ABB RAPID module: EGM_test_UDP.mod

MODULE EGM_test_UDP

    VAR egmident egmID1;
    VAR egmstate egmSt1;

    CONST egm_minmax egm_minmax_lin1:=[-1,1]; !in mm
    CONST egm_minmax egm_minmax_rot1:=[-2,2];! in degees
    CONST robtarget p20:=[[400,-300,100],[0,-1,0,0],[-1,0,1,0],[9E9,9E9,9E9,9E9,9E9,9E9]];

    PERS tooldata UISpenholder:=[TRUE,[[0,0,114.25],[1,0,0,0]],[1,[-0.095984607,0.082520613,38.69176324],[1,0,0,0],0,0,0]];
    PERS tooldata ToolOfLove:=[TRUE,[[0.015258,-0.149222,106.919],[0.999048,0.043619,0,0]],[1,[0,0,0.1],[1,0,0,0],0,0,0]];

    VAR pose posecorTable:=[[0,0,0],[1,0,0,0]];
    VAR pose posesenTable:=[[0,0,0],[1,0,0,0]];

    VAR speeddata speeddata0:=[500,500,5000,1000];


    PROC main()
        ! Move to start position. Fine point is demanded.
        MoveJ p20,speeddata0,fine,ToolOfLove;
        testuc_UDP;
    ENDPROC


    PROC testuc_UDP()
        EGMReset egmID1;
        EGMGetId egmID1;
        egmSt1 := EGMGetState(egmID1);
        TPWrite "EGM state: "\Num := egmSt1;

        IF egmSt1 <= EGM_STATE_CONNECTED THEN
            ! Set up the EGM data source: UdpUc server using device "EGMsensor:"and configuration "default"
            EGMSetupUC ROB_1, egmID1, "default", "EGMSensor:" \pose;
        ENDIF

        !Which program to run
        runEGM;

        IF egmSt1 = EGM_STATE_CONNECTED THEN
            TPWrite "Reset EGM instance egmID1";
            EGMReset egmID1;
        ENDIF
    ENDPROC


    PROC runEGM()
        EGMActPose egmID1\Tool:=ToolOfLove \WObj:=wobj0, posecorTable,EGM_FRAME_WOBJ, posesenTable, EGM_FRAME_WOBJ
        \x:=egm_minmax_lin1 \y:=egm_minmax_lin1 \z:=egm_minmax_lin1
        \rx:=egm_minmax_rot1 \ry:=egm_minmax_rot1 \rz:=egm_minmax_rot1\LpFilter:=2\Samplerate:=4\MaxSpeedDeviation:= 40;

        EGMRunPose egmID1, EGM_STOP_RAMP_DOWN\x \y \z\CondTime:=20 \RampInTime:=0.05\RampOutTime:=0.5;
        egmSt1:=EGMGetState(egmID1);

        ERROR

            IF ERRNO = ERR_UDPUC_COMM THEN !In case the computer stops sending positions
                TPWrite "The computer stoped sending corrdinates";
                EXIT;
            ENDIF
    ENDPROC

ENDMODULE
